{attribute 'GeneratedUsingTerminal: EL3202-0000-0016'}
{attribute addProperty BoxType "EL3202-0000-0016"}
{attribute addProperty Id "EtcSlaveTerminalBaseRTD_Inputs_Channel_1AT %I*RTD_Inputs_Channel_EA9DF21E9RTD_Inputs_Channel_2AT %I*RTD_Inputs_Channel_EA9DF21E9WcStateAT %I*WcState_9091E0EB2InfoDataAT %I*InfoData_32EB74EA10"}
{attribute addProperty CRC "1234443540"}
{attribute addProperty Size "30"}
TYPE EL3202_49941D14 EXTENDS EtcSlaveTerminalBase :
STRUCT
	{attribute addProperty Name "RTD_Inputs_Channel_1"}
	RTD_Inputs_Channel_1 : RTD_Inputs_Channel_EA9DF21E;
	{attribute addProperty Name "RTD_Inputs_Channel_2"}
	RTD_Inputs_Channel_2 : RTD_Inputs_Channel_EA9DF21E;
	{attribute addProperty Name "WcState"}
	WcState : WcState_9091E0EB;
	{attribute addProperty Name "InfoData"}
	InfoData : InfoData_32EB74EA;
END_STRUCT
END_TYPE

(* stored: Version 1.2.0.0, ProductVersion 3.1.4024.9
   DUT EL3202_49941D14: Id {79a8fe43-390f-4b7d-bf6a-1a5113683de9} *)
